TYPE ST_AlarmValue :
STRUCT
	Last_Alarm_Value:	REAL;
END_STRUCT
END_TYPE

(* stored: Version 1.1.0.1, ProductVersion 3.1.4020.6
   DUT ST_AlarmValue: Id {59947e1d-5de1-457f-811b-c80000c7f531} *)
